// Mitsubishi GX Works2 project: Ex02   PLC: Q02/Q02H

PROGRAM MAIN
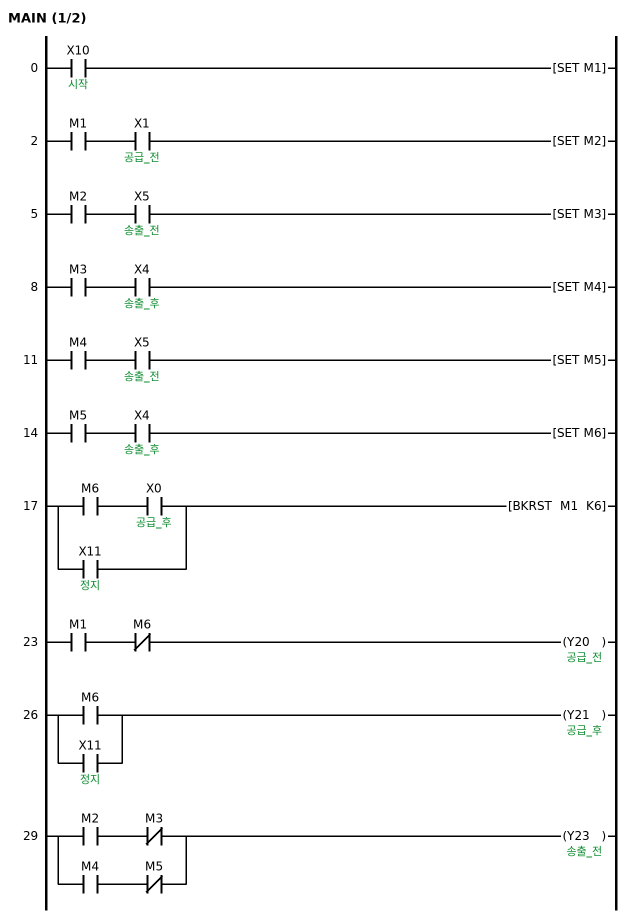
0     LD      X10  ; 시작
      SET     M1
2     LD      M1
      AND     X1  ; 공급_전
      SET     M2
5     LD      M2
      AND     X5  ; 송출_전
      SET     M3
8     LD      M3
      AND     X4  ; 송출_후
      SET     M4
11    LD      M4
      AND     X5  ; 송출_전
      SET     M5
14    LD      M5
      AND     X4  ; 송출_후
      SET     M6
17    LD      M6
      AND     X0  ; 공급_후
      OR      X11  ; 정지
      BKRST   M1 K6
23    LD      M1
      ANI     M6
      OUT     Y20  ; 공급_전
26    LD      M6
      OR      X11  ; 정지
      OUT     Y21  ; 공급_후
29    LD      M2
      ANI     M3
      LD      M4
      ANI     M5
      ORB
      OUT     Y23  ; 송출_전
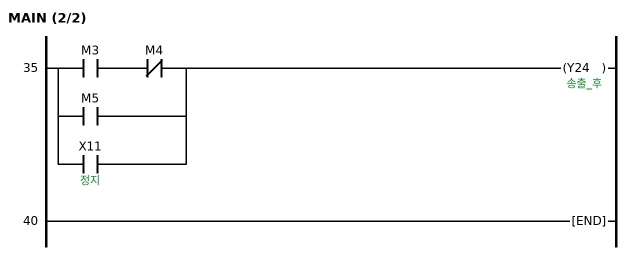
35    LD      M3
      ANI     M4
      OR      M5
      OR      X11  ; 정지
      OUT     Y24  ; 송출_후
40    END
END_PROGRAM

// device comments not shown above
X2  ; 드릴_상
X3  ; 드릴_하
X6  ; 배출_후
X7  ; 배출_전
X0A  ; 시작
X0B  ; 정지
Y22  ; 드릴_하강
Y25  ; 배출_전
Y26  ; 배출_후
